// TIA Portal V17 export
// export: Created 2024-08-20T10:59:38.6455385Z, ExportSetting WithDefaults, DisplayName Totally Integrated Automation Portal, DisplayVersion V17 Update 4, DisplayName TIA Portal Openness, DisplayVersion V17 Update 4, DisplayName TIA Portal Version Control Interface, DisplayVersion V17, DisplayName STEP 7 Professional, DisplayVersion V17 Update 4, DisplayName STEP 7 Safety, DisplayVersion V17, DisplayName WinCC Advanced, DisplayVersion V17 Update 4
FUNCTION_BLOCK "ROD2"   // FB205, LAD
TITLE = RODÍZIO DE 2 GRUPOS
{ S7_Optimized_Access := 'FALSE' }
VERSION : 0.1
// stored: AutoNumber false, IsIECCheckEnabled false, SetENOAutomatically false, UDAEnableTagReadback false
   VAR_INPUT
      G1OK : Bool;   // GRUPO EM CONDIÇÕES DE OPERAÇÃO
      G2OK : Bool;   // GRUPO EM CONDIÇÕES DE OPERAÇÃO
      G1L : Bool;   // GRUPO LIGADO
      G2L : Bool;   // GRUPO LIGADO
      TEROD : Int;   // TEMPOPARA RODÍZIO DAS BOMBAS
      LIGP : Bool;   // LIGA BOMBA PRINCIPAL
      LIGC1 : Bool;   // LIGA BOMBA COMPLEMENTAR 1
      DESAB : Bool;   // DESABILITA FUNCIONAMENTO DOS GRUPOS
      T1S : Bool;   // PULSO A CADA 1 SEGUNDO
      DESAB_PART : Bool;   // DESABILITA RODIZIO POR PARTIDA
   END_VAR
   VAR_OUTPUT
      G1P : Bool;   // GRUPO 1 SELECIONADO COMO PRINCIPAL
      G2P : Bool;   // GRUPO 2 SELECIONADO COMO PRINCIPAL
      G1C1 : Bool;   // GRUPO 1 SELECIONADO COMO COMPLEMENTAR 1
      G2C1 : Bool;   // GRUPO 2 SELECIONADO COMO COMPLEMENTAR 1
      LG1 : Bool;   // LIGA GRUPO 1
      LG2 : Bool;   // LIGA GRUPO 2
   END_VAR
   VAR_IN_OUT
      TOG1P : DInt;   // TEMPO DE OPERAÇÃO GRUPO 1
      TOG2P : DInt;   // TEMPO DE OPERAÇÃO GRUPO 2
      TEOKG1 : Real;   // TEMPO OK GRUPO 1
      TEOKG2 : Real;   // TEMPO OK GRUPO 2
   END_VAR
   VAR DB_SPECIFIC
      GR1SELP : Bool;   // SELECIONADO COMO PRINCIPAL
      GR2SELP : Bool;   // SELECIONADO COMO PRINCIPAL
      GR1SELC1 : Bool;   // SELECIONADO COMO COMPLEMENTAR 1
      GR2SELC1 : Bool;   // SELECIONADO COMO COMPLEMENTAR 1
      PS1SG1 : Bool;   // AUXILIAR DE PULSO
      PS1SG2 : Bool;   // AUXILIAR DE PULSO
      PS1 : Bool;   // AUXILIAR DE PULSO
      PS2 : Bool;   // AUXILIAR DE PULSO
      FIMTEG1 : Bool;   // FIM DO TEMPO DE EXISTÊNCIA DO GRUPO 1
      FIMTEG2 : Bool;   // FIM DO TEMPO DE EXISTÊNCIA DO GRUPO 2
      SDESG1 : Bool;   // SOLICITAÇÃO DE DESLIGAMENTO
      SDESG2 : Bool;   // SOLICITAÇÃO DE DESLIGAMENTO
      GPL : Bool;   // GRUPO PRINCIPAL LIGADO
      GC1L : Bool;   // GRUPO COMPLEMENTAR 1 LIGADO
      SO_L : Bool;   // SOLICITAÇÃO DE PARTIDA
      SO_D : Bool;   // SOLICITAÇÃO DE DESLIGAMENTO
      RTEOPG1 : Bool;   // RESET TEMPO OK
      RTEOPG2 : Bool;   // RESET TEMPO OK
      TON1 { S7_SetPoint := 'True'} : TON_TIME;   // TEMPORIZADOR
      TON2 { S7_SetPoint := 'True'} : TON_TIME;   // TEMPORIZADOR
      TSDG1 { S7_SetPoint := 'True'} : TON_TIME;   // TEMPORIZADOR
      TSDG2 { S7_SetPoint := 'True'} : TON_TIME;   // TEMPORIZADOR
   END_VAR
   VAR_TEMP
      PRI12 : Bool;   // PRIORIDADE GRUPO 1
      TMROD : DInt;   // TEMPO DE RODIZIO
      TEROD_DI : DInt;   // TEMPO DE RODIZIO
      NGS : Int;   // NÚMERO DE GRUPOS SOLICITADOS
      NGF : Int;   // NÚMERO DE GRUPOS FUNCIONANDO
      AUX01 : Int;   // AUXILIAR UTILIZADO NA LÓGICA
      AUX02 : Int;   // AUXILIAR UTILIZADO NA LÓGICA
      AUX03 : Int;   // AUXILIAR UTILIZADO NA LÓGICA
      AUX04 : Int;   // AUXILIAR UTILIZADO NA LÓGICA
      AUX05 : Bool;   // AUXILIAR UTILIZADO NA LÓGICA
      AUX06 : Bool;   // AUXILIAR UTILIZADO NA LÓGICA
      ETT1 : Time;   // EFETIVO DO TEMPORIZADOR
      ETT2 : Time;   // EFETIVO DO TEMPORIZADOR
      ETTSDG2 : Time;   // EFETIVO DO TEMPORIZADOR
      ETTSDG1 : Time;   // EFETIVO DO TEMPORIZADOR
   END_VAR
   VAR_TEMP   // added for the SCL form of the ladder/FBD networks
      _w1 : Bool;
   END_VAR
BEGIN

REGION Network 1: CONVERSÃO DO SETPOINT DE TEMPO DE RODÍZIO
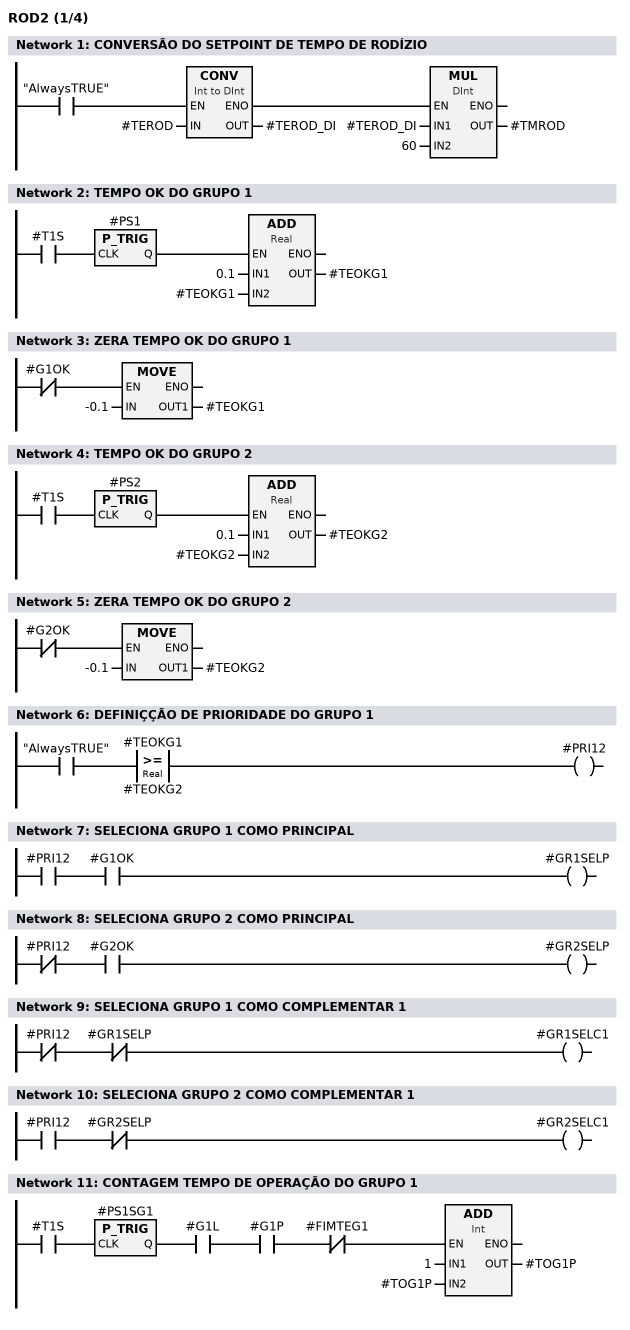
   RUNG wire#powerrail
      Contact( "AlwaysTRUE" )
      { S7_Templates := "[SrcType := Int, DestType := DInt]" } Convert(in := #TEROD, out => #TEROD_DI)
      { S7_Templates := "SrcType := DInt"; S7_GenerateENO := "TRUE" } Mul(in1 := #TEROD_DI, in2 := 60, out => #TMROD)
   END_RUNG
   // the same network as SCL:
   IF "AlwaysTRUE" THEN
       #TEROD_DI := INT_TO_DINT(#TEROD);
       #TMROD := #TEROD_DI * 60;
   END_IF;
END_REGION

REGION Network 2: TEMPO OK DO GRUPO 1
   RUNG wire#powerrail
      Contact( #T1S )
      P_Trig( #PS1 )
      { S7_Templates := "SrcType := Real"; S7_GenerateENO := "TRUE" } Add(in1 := 0.1, in2 := #TEOKG1, out => #TEOKG1)
   END_RUNG
   // the same network as SCL:
   #_w1 := #T1S AND NOT #PS1;   // rising edge
   #PS1 := #T1S;
   IF #_w1 THEN #TEOKG1 := 0.1 + #TEOKG1; END_IF;
END_REGION

REGION Network 3: ZERA TEMPO OK DO GRUPO 1
   RUNG wire#powerrail
      I_Contact( #G1OK )
      { S7_GenerateENO := "TRUE" } Move(in := -0.1, out1 => #TEOKG1)
   END_RUNG
   // the same network as SCL:
   IF NOT #G1OK THEN #TEOKG1 := -0.1; END_IF;
END_REGION

REGION Network 4: TEMPO OK DO GRUPO 2
   RUNG wire#powerrail
      Contact( #T1S )
      P_Trig( #PS2 )
      { S7_Templates := "SrcType := Real"; S7_GenerateENO := "TRUE" } Add(in1 := 0.1, in2 := #TEOKG2, out => #TEOKG2)
   END_RUNG
   // the same network as SCL:
   #_w1 := #T1S AND NOT #PS2;   // rising edge
   #PS2 := #T1S;
   IF #_w1 THEN #TEOKG2 := 0.1 + #TEOKG2; END_IF;
END_REGION

REGION Network 5: ZERA TEMPO OK DO GRUPO 2
   RUNG wire#powerrail
      I_Contact( #G2OK )
      { S7_GenerateENO := "TRUE" } Move(in := -0.1, out1 => #TEOKG2)
   END_RUNG
   // the same network as SCL:
   IF NOT #G2OK THEN #TEOKG2 := -0.1; END_IF;
END_REGION

REGION Network 6: DEFINIÇÇÃO DE PRIORIDADE DO GRUPO 1
   RUNG wire#powerrail
      Contact( "AlwaysTRUE" )
      { S7_Templates := "SrcType := Real" } GE_Contact(in1 := #TEOKG1, in2 := #TEOKG2)
      Coil( #PRI12 )
   END_RUNG
   // the same network as SCL:
   #PRI12 := "AlwaysTRUE" AND (#TEOKG1 >= #TEOKG2);
END_REGION

REGION Network 7: SELECIONA GRUPO 1 COMO PRINCIPAL
   RUNG wire#powerrail
      Contact( #PRI12 )
      Contact( #G1OK )
      Coil( #GR1SELP )
   END_RUNG
   // the same network as SCL:
   #GR1SELP := #PRI12 AND #G1OK;
END_REGION

REGION Network 8: SELECIONA GRUPO 2 COMO PRINCIPAL
   RUNG wire#powerrail
      I_Contact( #PRI12 )
      Contact( #G2OK )
      Coil( #GR2SELP )
   END_RUNG
   // the same network as SCL:
   #GR2SELP := NOT #PRI12 AND #G2OK;
END_REGION

REGION Network 9: SELECIONA GRUPO 1 COMO COMPLEMENTAR 1
   RUNG wire#powerrail
      I_Contact( #PRI12 )
      I_Contact( #GR1SELP )
      Coil( #GR1SELC1 )
   END_RUNG
   // the same network as SCL:
   #GR1SELC1 := NOT #PRI12 AND NOT #GR1SELP;
END_REGION

REGION Network 10: SELECIONA GRUPO 2 COMO COMPLEMENTAR 1
   RUNG wire#powerrail
      Contact( #PRI12 )
      I_Contact( #GR2SELP )
      Coil( #GR2SELC1 )
   END_RUNG
   // the same network as SCL:
   #GR2SELC1 := #PRI12 AND NOT #GR2SELP;
END_REGION

REGION Network 11: CONTAGEM TEMPO DE OPERAÇÃO DO GRUPO 1
   RUNG wire#powerrail
      Contact( #T1S )
      P_Trig( #PS1SG1 )
      Contact( #G1L )
      Contact( #G1P )
      I_Contact( #FIMTEG1 )
      { S7_Templates := "SrcType := Int"; S7_GenerateENO := "TRUE" } Add(in1 := 1, in2 := #TOG1P, out => #TOG1P)
   END_RUNG
   // the same network as SCL:
   #_w1 := #T1S AND NOT #PS1SG1;   // rising edge
   #PS1SG1 := #T1S;
   IF #_w1 AND #G1L AND #G1P AND NOT #FIMTEG1 THEN #TOG1P := 1 + #TOG1P; END_IF;
END_REGION

REGION Network 12: TEMPO DE OPERAÇÃO ATINGIDO
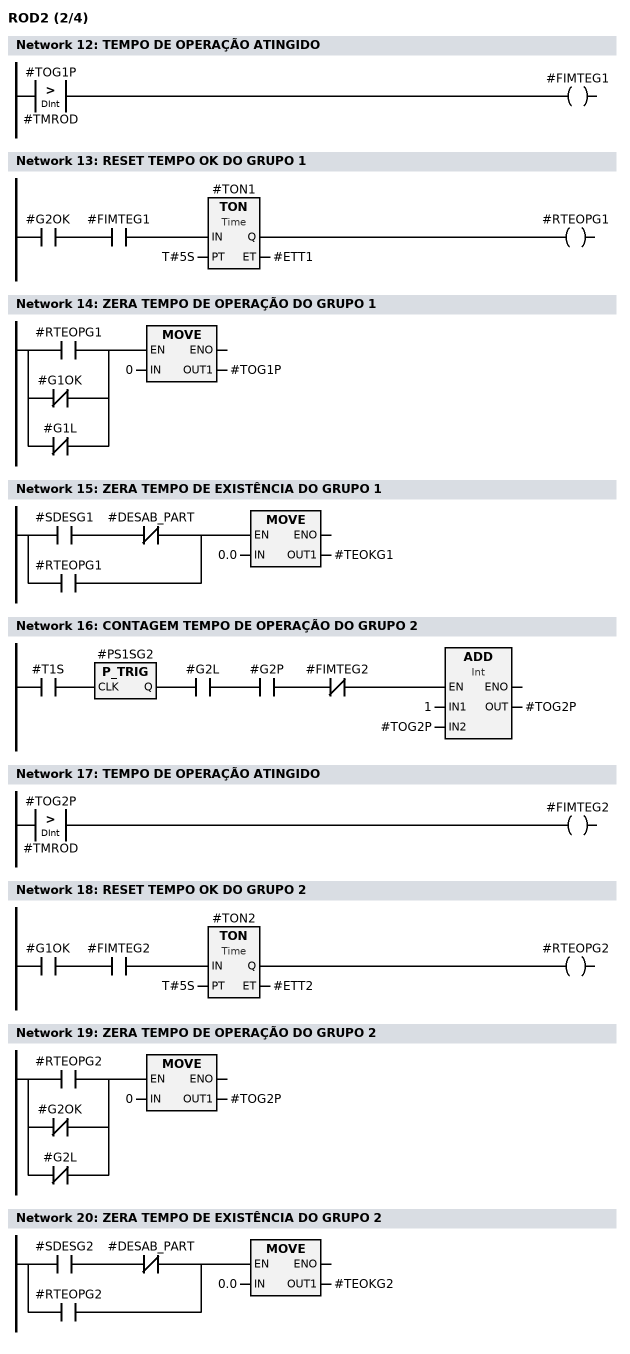
   RUNG wire#powerrail
      { S7_Templates := "SrcType := DInt" } GT_Contact(in1 := #TOG1P, in2 := #TMROD)
      Coil( #FIMTEG1 )
   END_RUNG
   // the same network as SCL:
   #FIMTEG1 := #TOG1P > #TMROD;
END_REGION

REGION Network 13: RESET TEMPO OK DO GRUPO 1
   RUNG wire#powerrail
      Contact( #G2OK )
      Contact( #FIMTEG1 )
      { S7_Templates := "time_type := Time" } #TON1.TON(pt := T#5S, et => #ETT1)
      Coil( #RTEOPG1 )
   END_RUNG
   // the same network as SCL:
   #TON1(IN := #G2OK AND #FIMTEG1, PT := T#5S, ET => #ETT1);   // TON
   #RTEOPG1 := #TON1.Q;
END_REGION

REGION Network 14: ZERA TEMPO DE OPERAÇÃO DO GRUPO 1
   RUNG wire#powerrail
      Contact( #RTEOPG1 )
      wire#w1
      { S7_GenerateENO := "TRUE" } Move(in := 0, out1 => #TOG1P)
   END_RUNG
   RUNG wire#powerrail
      I_Contact( #G1OK )
   END_RUNG wire#w1
   RUNG wire#powerrail
      I_Contact( #G1L )
   END_RUNG wire#w1
   // the same network as SCL:
   IF #RTEOPG1 OR NOT #G1OK OR NOT #G1L THEN #TOG1P := 0; END_IF;
END_REGION

REGION Network 15: ZERA TEMPO DE EXISTÊNCIA DO GRUPO 1
   RUNG wire#powerrail
      Contact( #SDESG1 )
      I_Contact( #DESAB_PART )
      wire#w1
      { S7_GenerateENO := "TRUE" } Move(in := 0.0, out1 => #TEOKG1)
   END_RUNG
   RUNG wire#powerrail
      Contact( #RTEOPG1 )
   END_RUNG wire#w1
   // the same network as SCL:
   IF (#SDESG1 AND NOT #DESAB_PART) OR #RTEOPG1 THEN #TEOKG1 := 0.0; END_IF;
END_REGION

REGION Network 16: CONTAGEM TEMPO DE OPERAÇÃO DO GRUPO 2
   RUNG wire#powerrail
      Contact( #T1S )
      P_Trig( #PS1SG2 )
      Contact( #G2L )
      Contact( #G2P )
      I_Contact( #FIMTEG2 )
      { S7_Templates := "SrcType := Int"; S7_GenerateENO := "TRUE" } Add(in1 := 1, in2 := #TOG2P, out => #TOG2P)
   END_RUNG
   // the same network as SCL:
   #_w1 := #T1S AND NOT #PS1SG2;   // rising edge
   #PS1SG2 := #T1S;
   IF #_w1 AND #G2L AND #G2P AND NOT #FIMTEG2 THEN #TOG2P := 1 + #TOG2P; END_IF;
END_REGION

REGION Network 17: TEMPO DE OPERAÇÃO ATINGIDO
   RUNG wire#powerrail
      { S7_Templates := "SrcType := DInt" } GT_Contact(in1 := #TOG2P, in2 := #TMROD)
      Coil( #FIMTEG2 )
   END_RUNG
   // the same network as SCL:
   #FIMTEG2 := #TOG2P > #TMROD;
END_REGION

REGION Network 18: RESET TEMPO OK DO GRUPO 2
   RUNG wire#powerrail
      Contact( #G1OK )
      Contact( #FIMTEG2 )
      { S7_Templates := "time_type := Time" } #TON2.TON(pt := T#5S, et => #ETT2)
      Coil( #RTEOPG2 )
   END_RUNG
   // the same network as SCL:
   #TON2(IN := #G1OK AND #FIMTEG2, PT := T#5S, ET => #ETT2);   // TON
   #RTEOPG2 := #TON2.Q;
END_REGION

REGION Network 19: ZERA TEMPO DE OPERAÇÃO DO GRUPO 2
   RUNG wire#powerrail
      Contact( #RTEOPG2 )
      wire#w1
      { S7_GenerateENO := "TRUE" } Move(in := 0, out1 => #TOG2P)
   END_RUNG
   RUNG wire#powerrail
      I_Contact( #G2OK )
   END_RUNG wire#w1
   RUNG wire#powerrail
      I_Contact( #G2L )
   END_RUNG wire#w1
   // the same network as SCL:
   IF #RTEOPG2 OR NOT #G2OK OR NOT #G2L THEN #TOG2P := 0; END_IF;
END_REGION

REGION Network 20: ZERA TEMPO DE EXISTÊNCIA DO GRUPO 2
   RUNG wire#powerrail
      Contact( #SDESG2 )
      I_Contact( #DESAB_PART )
      wire#w1
      { S7_GenerateENO := "TRUE" } Move(in := 0.0, out1 => #TEOKG2)
   END_RUNG
   RUNG wire#powerrail
      Contact( #RTEOPG2 )
   END_RUNG wire#w1
   // the same network as SCL:
   IF (#SDESG2 AND NOT #DESAB_PART) OR #RTEOPG2 THEN #TEOKG2 := 0.0; END_IF;
END_REGION

REGION Network 21: SELEÇÃO GRUPO 1 COMO PRINCIPAL
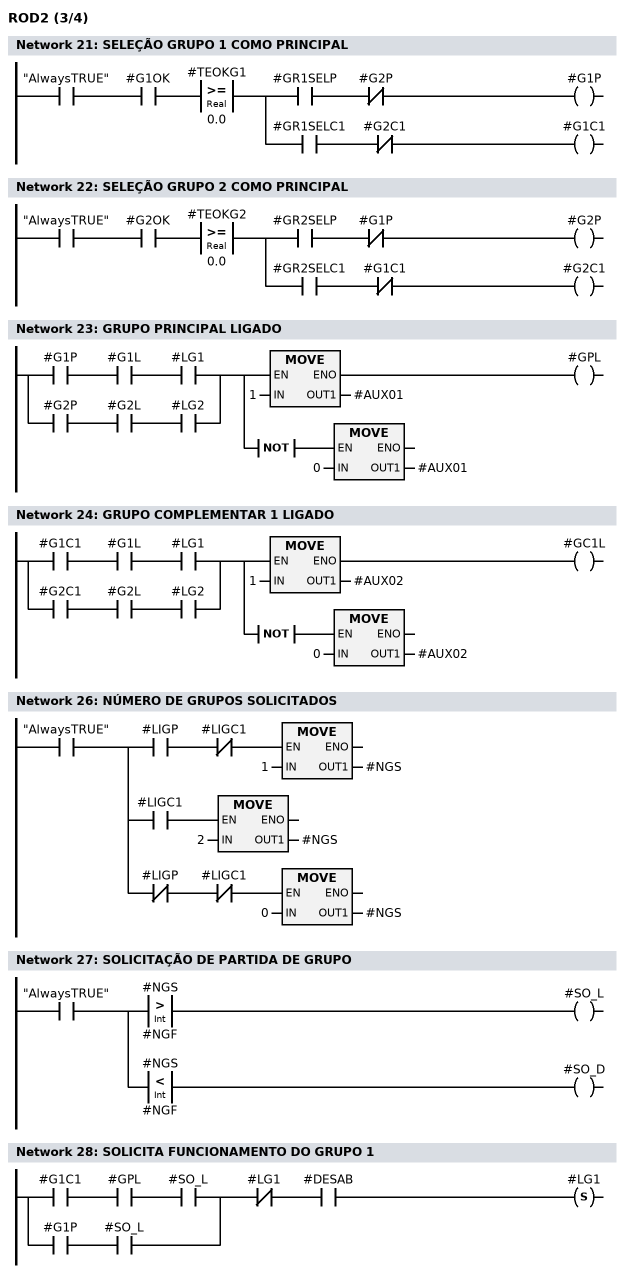
   RUNG wire#powerrail
      Contact( "AlwaysTRUE" )
      Contact( #G1OK )
      { S7_Templates := "SrcType := Real" } GE_Contact(in1 := #TEOKG1, in2 := 0.0)
      wire#w1
      Contact( #GR1SELP )
      I_Contact( #G2P )
      Coil( #G1P )
   END_RUNG
   RUNG wire#w1
      Contact( #GR1SELC1 )
      I_Contact( #G2C1 )
      Coil( #G1C1 )
   END_RUNG
   // the same network as SCL:
   #_w1 := "AlwaysTRUE" AND #G1OK AND (#TEOKG1 >= 0.0);
   #G1P := #_w1 AND #GR1SELP AND NOT #G2P;
   #G1C1 := #_w1 AND #GR1SELC1 AND NOT #G2C1;
END_REGION

REGION Network 22: SELEÇÃO GRUPO 2 COMO PRINCIPAL
   RUNG wire#powerrail
      Contact( "AlwaysTRUE" )
      Contact( #G2OK )
      { S7_Templates := "SrcType := Real" } GE_Contact(in1 := #TEOKG2, in2 := 0.0)
      wire#w1
      Contact( #GR2SELP )
      I_Contact( #G1P )
      Coil( #G2P )
   END_RUNG
   RUNG wire#w1
      Contact( #GR2SELC1 )
      I_Contact( #G1C1 )
      Coil( #G2C1 )
   END_RUNG
   // the same network as SCL:
   #_w1 := "AlwaysTRUE" AND #G2OK AND (#TEOKG2 >= 0.0);
   #G2P := #_w1 AND #GR2SELP AND NOT #G1P;
   #G2C1 := #_w1 AND #GR2SELC1 AND NOT #G1C1;
END_REGION

REGION Network 23: GRUPO PRINCIPAL LIGADO
   RUNG wire#powerrail
      Contact( #G1P )
      Contact( #G1L )
      Contact( #LG1 )
      wire#w1
      { S7_GenerateENO := "TRUE" } Move(in := 1, out1 => #AUX01)
      Coil( #GPL )
   END_RUNG
   RUNG wire#powerrail
      Contact( #G2P )
      Contact( #G2L )
      Contact( #LG2 )
   END_RUNG wire#w1
   RUNG wire#w1
      Not()
      { S7_GenerateENO := "TRUE" } Move(in := 0, out1 => #AUX01)
   END_RUNG
   // the same network as SCL:
   // ENO of a box is taken as its EN; it also drops when the box reports an error
   #_w1 := (#G1P AND #G1L AND #LG1) OR (#G2P AND #G2L AND #LG2);
   IF #_w1 THEN #AUX01 := 1; END_IF;
   #GPL := #_w1;
   IF NOT #_w1 THEN #AUX01 := 0; END_IF;
END_REGION

REGION Network 24: GRUPO COMPLEMENTAR 1 LIGADO
   RUNG wire#powerrail
      Contact( #G1C1 )
      Contact( #G1L )
      Contact( #LG1 )
      wire#w1
      { S7_GenerateENO := "TRUE" } Move(in := 1, out1 => #AUX02)
      Coil( #GC1L )
   END_RUNG
   RUNG wire#powerrail
      Contact( #G2C1 )
      Contact( #G2L )
      Contact( #LG2 )
   END_RUNG wire#w1
   RUNG wire#w1
      Not()
      { S7_GenerateENO := "TRUE" } Move(in := 0, out1 => #AUX02)
   END_RUNG
   // the same network as SCL:
   // ENO of a box is taken as its EN; it also drops when the box reports an error
   #_w1 := (#G1C1 AND #G1L AND #LG1) OR (#G2C1 AND #G2L AND #LG2);
   IF #_w1 THEN #AUX02 := 1; END_IF;
   #GC1L := #_w1;
   IF NOT #_w1 THEN #AUX02 := 0; END_IF;
END_REGION

NETWORK
TITLE = NÚMERO DE GRUPOS FUNCIONANDO

      L     #AUX01;
      L     #AUX02;
      +I;
      T     #NGF;

REGION Network 26: NÚMERO DE GRUPOS SOLICITADOS
   RUNG wire#powerrail
      Contact( "AlwaysTRUE" )
      wire#w1
      Contact( #LIGP )
      I_Contact( #LIGC1 )
      { S7_GenerateENO := "TRUE" } Move(in := 1, out1 => #NGS)
   END_RUNG
   RUNG wire#w1
      Contact( #LIGC1 )
      { S7_GenerateENO := "TRUE" } Move(in := 2, out1 => #NGS)
   END_RUNG
   RUNG wire#w1
      I_Contact( #LIGP )
      I_Contact( #LIGC1 )
      { S7_GenerateENO := "TRUE" } Move(in := 0, out1 => #NGS)
   END_RUNG
   // the same network as SCL:
   IF "AlwaysTRUE" AND #LIGP AND NOT #LIGC1 THEN #NGS := 1; END_IF;
   IF "AlwaysTRUE" AND #LIGC1 THEN #NGS := 2; END_IF;
   IF "AlwaysTRUE" AND NOT #LIGP AND NOT #LIGC1 THEN #NGS := 0; END_IF;
END_REGION

REGION Network 27: SOLICITAÇÃO DE PARTIDA DE GRUPO
   RUNG wire#powerrail
      Contact( "AlwaysTRUE" )
      wire#w1
      { S7_Templates := "SrcType := Int" } GT_Contact(in1 := #NGS, in2 := #NGF)
      Coil( #SO_L )
   END_RUNG
   RUNG wire#w1
      { S7_Templates := "SrcType := Int" } LT_Contact(in1 := #NGS, in2 := #NGF)
      Coil( #SO_D )
   END_RUNG
   // the same network as SCL:
   #SO_L := "AlwaysTRUE" AND (#NGS > #NGF);
   #SO_D := "AlwaysTRUE" AND (#NGS < #NGF);
END_REGION

REGION Network 28: SOLICITA FUNCIONAMENTO DO GRUPO 1
   RUNG wire#powerrail
      Contact( #G1C1 )
      Contact( #GPL )
      Contact( #SO_L )
      wire#w1
      I_Contact( #LG1 )
      Contact( #DESAB )
      S_Coil( #LG1 )
   END_RUNG
   RUNG wire#powerrail
      Contact( #G1P )
      Contact( #SO_L )
   END_RUNG wire#w1
   // the same network as SCL:
   IF ((#G1C1 AND #GPL AND #SO_L) OR (#G1P AND #SO_L)) AND NOT #LG1 AND #DESAB THEN #LG1 := TRUE; END_IF;
END_REGION

REGION Network 29: SOLICITA FUNCIONAMENTO DO GRUPO 2
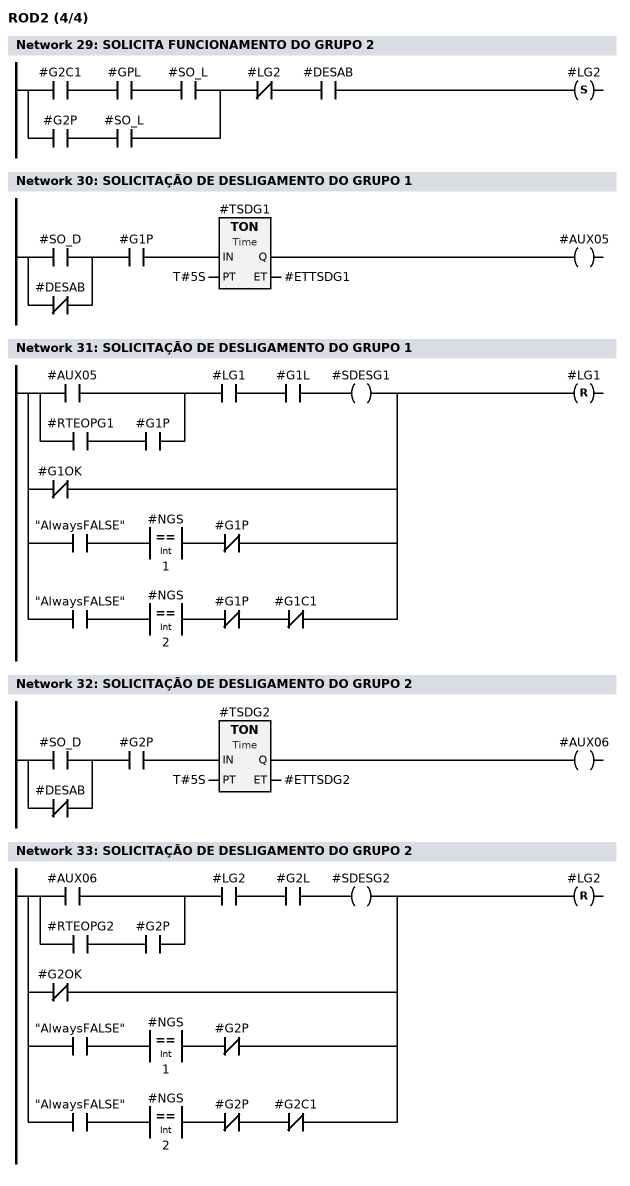
   RUNG wire#powerrail
      Contact( #G2C1 )
      Contact( #GPL )
      Contact( #SO_L )
      wire#w1
      I_Contact( #LG2 )
      Contact( #DESAB )
      S_Coil( #LG2 )
   END_RUNG
   RUNG wire#powerrail
      Contact( #G2P )
      Contact( #SO_L )
   END_RUNG wire#w1
   // the same network as SCL:
   IF ((#G2C1 AND #GPL AND #SO_L) OR (#G2P AND #SO_L)) AND NOT #LG2 AND #DESAB THEN #LG2 := TRUE; END_IF;
END_REGION

REGION Network 30: SOLICITAÇÃO DE DESLIGAMENTO DO GRUPO 1
   RUNG wire#powerrail
      Contact( #SO_D )
      wire#w1
      Contact( #G1P )
      { S7_Templates := "time_type := Time" } #TSDG1.TON(pt := T#5S, et => #ETTSDG1)
      Coil( #AUX05 )
   END_RUNG
   RUNG wire#powerrail
      I_Contact( #DESAB )
   END_RUNG wire#w1
   // the same network as SCL:
   #TSDG1(IN := (#SO_D OR NOT #DESAB) AND #G1P, PT := T#5S, ET => #ETTSDG1);   // TON
   #AUX05 := #TSDG1.Q;
END_REGION

REGION Network 31: SOLICITAÇÃO DE DESLIGAMENTO DO GRUPO 1
   RUNG wire#powerrail
      Contact( #AUX05 )
      wire#w1
      Contact( #LG1 )
      Contact( #G1L )
      Coil( #SDESG1 )
      wire#w2
      R_Coil( #LG1 )
   END_RUNG
   RUNG wire#powerrail
      Contact( #RTEOPG1 )
      Contact( #G1P )
   END_RUNG wire#w1
   RUNG wire#powerrail
      I_Contact( #G1OK )
   END_RUNG wire#w2
   RUNG wire#powerrail
      Contact( "AlwaysFALSE" )
      { S7_Templates := "SrcType := Int" } EQ_Contact(in1 := #NGS, in2 := 1)
      I_Contact( #G1P )
   END_RUNG wire#w2
   RUNG wire#powerrail
      Contact( "AlwaysFALSE" )
      { S7_Templates := "SrcType := Int" } EQ_Contact(in1 := #NGS, in2 := 2)
      I_Contact( #G1P )
      I_Contact( #G1C1 )
   END_RUNG wire#w2
   // the same network as SCL:
   #SDESG1 := (#AUX05 OR (#RTEOPG1 AND #G1P)) AND #LG1 AND #G1L;
   IF #SDESG1 OR NOT #G1OK OR ("AlwaysFALSE" AND (#NGS = 1) AND NOT #G1P) OR ("AlwaysFALSE" AND (#NGS = 2) AND NOT #G1P AND NOT #G1C1) THEN
       #LG1 := FALSE;
   END_IF;
END_REGION

REGION Network 32: SOLICITAÇÃO DE DESLIGAMENTO DO GRUPO 2
   RUNG wire#powerrail
      Contact( #SO_D )
      wire#w1
      Contact( #G2P )
      { S7_Templates := "time_type := Time" } #TSDG2.TON(pt := T#5S, et => #ETTSDG2)
      Coil( #AUX06 )
   END_RUNG
   RUNG wire#powerrail
      I_Contact( #DESAB )
   END_RUNG wire#w1
   // the same network as SCL:
   #TSDG2(IN := (#SO_D OR NOT #DESAB) AND #G2P, PT := T#5S, ET => #ETTSDG2);   // TON
   #AUX06 := #TSDG2.Q;
END_REGION

REGION Network 33: SOLICITAÇÃO DE DESLIGAMENTO DO GRUPO 2
   RUNG wire#powerrail
      Contact( #AUX06 )
      wire#w1
      Contact( #LG2 )
      Contact( #G2L )
      Coil( #SDESG2 )
      wire#w2
      R_Coil( #LG2 )
   END_RUNG
   RUNG wire#powerrail
      Contact( #RTEOPG2 )
      Contact( #G2P )
   END_RUNG wire#w1
   RUNG wire#powerrail
      I_Contact( #G2OK )
   END_RUNG wire#w2
   RUNG wire#powerrail
      Contact( "AlwaysFALSE" )
      { S7_Templates := "SrcType := Int" } EQ_Contact(in1 := #NGS, in2 := 1)
      I_Contact( #G2P )
   END_RUNG wire#w2
   RUNG wire#powerrail
      Contact( "AlwaysFALSE" )
      { S7_Templates := "SrcType := Int" } EQ_Contact(in1 := #NGS, in2 := 2)
      I_Contact( #G2P )
      I_Contact( #G2C1 )
   END_RUNG wire#w2
   // the same network as SCL:
   #SDESG2 := (#AUX06 OR (#RTEOPG2 AND #G2P)) AND #LG2 AND #G2L;
   IF #SDESG2 OR NOT #G2OK OR ("AlwaysFALSE" AND (#NGS = 1) AND NOT #G2P) OR ("AlwaysFALSE" AND (#NGS = 2) AND NOT #G2P AND NOT #G2C1) THEN
       #LG2 := FALSE;
   END_IF;
END_REGION
END_FUNCTION_BLOCK
